FUNCTION_BLOCK Mc2MoveJogTask EXTENDS Mc2MotionTask IMPLEMENTS I_Mc2MotionJogTask
VAR
	McJog		  : Tc2_MC2.MC_Jog;
	_JogForward	  : BOOL;
	_JogBackwards : BOOL;
	_Mode		  : Tc2_MC2.E_JogMode;
	_Position	  : LREAL;
END_VAR

{attribute 'monitoring' := 'call'}
PROPERTY Busy : BOOL
GET
Busy := MCJog.Busy;
END_GET
END_PROPERTY

METHOD CyclicLogic
McJog(Axis		   := _Axis.Axis,
	  Velocity	   := _Axis.Velocity,
	  Acceleration := _Axis.Acceleration,
	  Deceleration := _Axis.Deceleration,
	  Jerk		   := _Axis.Jerk);
      
IF McJog.Error OR _Axis.Error THEN
    _JogForward := FALSE;
    _JogBackwards := FALSE;
END_IF
END_METHOD

{attribute 'monitoring' := 'call'}
PROPERTY Error : BOOL
GET
Error := MCJog.Error;
END_GET
END_PROPERTY

{attribute 'monitoring' := 'call'}
PROPERTY ErrorId : UDINT
GET
ErrorId := MCJog.ErrorID;
END_GET
END_PROPERTY

METHOD Execute : BOOL
McJog(Axis		   := _Axis.Axis,
	  JogForward   := _JogForward,
	  JogBackwards := _JogBackwards,
	  Mode		   := _Mode,
	  Position	   := _Position);
END_METHOD

PROPERTY JogBackwards : BOOL
SET
_JogBackwards := JogBackwards;
END_SET
END_PROPERTY

PROPERTY JogForward : BOOL
SET
_JogForward := JogForward;
END_SET
END_PROPERTY

PROPERTY Mode : E_JogMode
SET
_Mode := Mode;
END_SET
END_PROPERTY

PROPERTY Position : LREAL
SET
_Position := Position;
END_SET
END_PROPERTY

END_FUNCTION_BLOCK

(* stored: Version 1.1.0.1, ProductVersion 3.1.4026.20
   POU Mc2MoveJogTask: Id {949ec021-9e06-4765-b74e-0dd100d557b2}, SpecialFunc None
   Property Busy: Id {b72d5904-9bfc-4514-acb7-1f22fa0b534b}
   Get Get: Id {7d70124e-1302-4c1a-abdf-8e220863faef}
   Method CyclicLogic: Id {30bdeb88-7bd6-4b2f-96bd-ec1b2f7219a2}
   Property Error: Id {84420d75-ad24-4d3a-8cef-0d3144af0820}
   Get Get: Id {e11c98b5-4e50-4b50-b742-7461cd584d12}
   Property ErrorId: Id {95504fdc-fa04-4d67-815f-b0ed06f5a0cf}
   Get Get: Id {4baa563d-ded1-4b72-9ff7-9946736b121e}
   Method Execute: Id {4b27b5b6-b31f-4d84-b855-5827507dc4b4}
   Property JogBackwards: Id {d2b5dab1-f45a-4e3d-be2c-05d411cc1ef6}
   Set Set: Id {f0740fec-7256-4bea-9d26-8aa30207f2fe}
   Property JogForward: Id {81e7ed2d-2f35-4455-a04c-953404cc4d3c}
   Set Set: Id {8bc556cc-67e9-41b4-bd7d-472843338c61}
   Property Mode: Id {1fce2653-7463-4826-be32-f4cd665c43bd}
   Set Set: Id {528e85dc-b9a5-4a65-8e4d-5be74dc91129}
   Property Position: Id {093b613a-4624-4500-a07a-295591354775}
   Set Set: Id {5c8ab3e9-e9c8-40cc-a33e-b96060121f40} *)
